// TIA Portal V16 export
// export: Created 2020-05-03T18:29:29.4641173Z, ExportSetting WithDefaults, DisplayName Totally Integrated Automation Portal, DisplayVersion V16, DisplayName TIA Portal Version Control Interface, DisplayVersion V16, DisplayName TIA Portal Openness, DisplayVersion V16, DisplayName STEP 7 Professional, DisplayVersion V16, DisplayName STEP 7 Safety, DisplayVersion V16, DisplayName WinCC Unified SCADA Engineering System, DisplayVersion V16
VAR_GLOBAL   // PLC tag table "Default tag table"
   Example_1 AT %M0.0 : Bool;
   ExOut AT %Q0.0 : Bool;
END_VAR
